// TwinCAT 3 PLC project PLC1
// ProgramVersion: 3.1.4024.0
// libraries:
//   Tc2_Standard, * (Beckhoff Automation GmbH)
//   Tc2_System, * (Beckhoff Automation GmbH)
//   Tc3_Module, * (Beckhoff Automation GmbH)
// project tree:
//   GVLs/ GVL.TcGVL
//   / PlcTask.TcTTO
//   POUs/ MAIN.TcPOU
// real-time tasks:
//   TASK PlcTask: cycle T#10ms, priority 20, ADS port 350

CONFIGURATION PLC1
    RESOURCE PLC ON TwinCAT3
        TASK PlcTask(INTERVAL := T#10ms, PRIORITY := 20);
        PROGRAM MAIN WITH PlcTask : MAIN;
    END_RESOURCE
END_CONFIGURATION

// ---- GVLs/GVL.TcGVL
{attribute 'qualified_only'}
VAR_GLOBAL
	SinOfAngle : LREAL;
END_VAR

// ---- POUs/MAIN.TcPOU
PROGRAM MAIN
VAR
	AngleDeg : LREAL;
	AngleRad : LREAL;
END_VAR

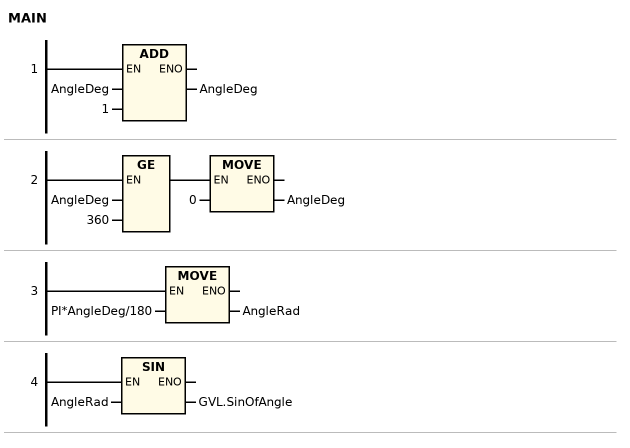
// NETWORK 1
AngleDeg := AngleDeg + 1;

// NETWORK 2
IF AngleDeg >= 360 THEN AngleDeg := 0; END_IF

// NETWORK 3
AngleRad := PI*AngleDeg/180;

// NETWORK 4
GVL.SinOfAngle := SIN(AngleRad);

END_PROGRAM
